    CONST robtarget rA_t486 := [[-156.188,32.3569,3418.1],[0.820893,-0.20476,-0.394721,0.358334],[1,0,2,0],[9E+09,9E+09,9E+09,9E+09,9E+09,9E+09]];
    CONST robtarget rB_t486 := [[608.123,552.232,3105.31],[0.872277,-0.183235,0.197016,-0.408341],[0,-2,0,0],[9E+09,9E+09,9E+09,9E+09,9E+09,9E+09]];
    CONST robtarget rB_t486_c5 := [[608.123,552.232,3105.31],[0.872277,-0.183235,0.197016,-0.408341],[0,0,0,0],[9E+09,9E+09,9E+09,9E+09,9E+09,9E+09]];
    CONST jointtarget jA_t486 := [[135,-13.9732,-69.2642,45,47.8597,225],[9E+09,9E+09,9E+09,9E+09,9E+09,9E+09]];
    CONST jointtarget jB_t486 := [[44.9992,-24.9745,-22.5996,-135.001,19.5471,44.9992],[9E+09,9E+09,9E+09,9E+09,9E+09,9E+09]];
    CONST jointtarget jBseed_t486 := [[44.9992,-24.9745,-22.5996,-135.001,19.5471,44.9992],[9E+09,9E+09,9E+09,9E+09,9E+09,9E+09]];

    CONST robtarget rA_t488 := [[-1759.7,-1640.61,1999.46],[0.855755,-0.00396172,-0.496397,0.145798],[-2,2,-1,0],[9E+09,9E+09,9E+09,9E+09,9E+09,9E+09]];
    CONST robtarget rB_t488 := [[478.399,-39.3809,2596.98],[0.780574,-0.0851872,0.494213,-0.373097],[-1,-1,-1,0],[9E+09,9E+09,9E+09,9E+09,9E+09,9E+09]];
    CONST robtarget rB_t488_c5 := [[478.399,-39.3809,2596.98],[0.780574,-0.0851872,0.494213,-0.373097],[0,0,0,0],[9E+09,9E+09,9E+09,9E+09,9E+09,9E+09]];
    CONST jointtarget jA_t488 := [[-135.001,22.0814,-22.3377,224.999,45.461,-45.001],[9E+09,9E+09,9E+09,9E+09,9E+09,9E+09]];
    CONST jointtarget jB_t488 := [[-0.000711459,-56.8981,12.0994,-45.0007,19.4775,-0.00071639],[9E+09,9E+09,9E+09,9E+09,9E+09,9E+09]];
    CONST jointtarget jBseed_t488 := [[-0.000711051,-56.8981,12.0994,-45.0007,19.4775,-0.000711051],[9E+09,9E+09,9E+09,9E+09,9E+09,9E+09]];

    CONST robtarget rA_t489 := [[478.399,-39.3809,2596.98],[0.780574,-0.0851872,0.494213,-0.373097],[-1,-1,-1,0],[9E+09,9E+09,9E+09,9E+09,9E+09,9E+09]];
    CONST robtarget rB_t489 := [[-73.1734,1033.07,3314.31],[0.0648344,0.215246,-0.280952,-0.933023],[1,-3,4,0],[9E+09,9E+09,9E+09,9E+09,9E+09,9E+09]];
    CONST robtarget rB_t489_c4 := [[-73.1734,1033.07,3314.31],[0.0648344,0.215246,-0.280952,-0.933023],[0,-4,0,0],[9E+09,9E+09,9E+09,9E+09,9E+09,9E+09]];
    CONST robtarget rB_t489_c5 := [[-73.1734,1033.07,3314.31],[0.0648344,0.215246,-0.280952,-0.933023],[0,0,0,0],[9E+09,9E+09,9E+09,9E+09,9E+09,9E+09]];
    CONST jointtarget jA_t489 := [[-0.000711459,-56.8981,12.0994,-45.0007,19.4775,-0.00071639],[9E+09,9E+09,9E+09,9E+09,9E+09,9E+09]];
    CONST jointtarget jB_t489 := [[90.0008,-2.94625,-53.5374,-269.999,25.9816,360.001],[9E+09,9E+09,9E+09,9E+09,9E+09,9E+09]];
    CONST jointtarget jBseed_t489 := [[90.0008,-2.94625,-53.5374,-269.999,25.9816,360.001],[9E+09,9E+09,9E+09,9E+09,9E+09,9E+09]];

    CONST robtarget rA_t490 := [[-73.1734,1033.07,3314.31],[0.0648344,0.215246,-0.280952,-0.933023],[1,-3,4,0],[9E+09,9E+09,9E+09,9E+09,9E+09,9E+09]];
    CONST robtarget rB_t490 := [[1761.71,1761.73,978.083],[0.626552,-0.67896,0.281238,-0.25952],[0,2,1,0],[9E+09,9E+09,9E+09,9E+09,9E+09,9E+09]];
    CONST robtarget rB_t490_c4 := [[1761.71,1761.73,978.083],[0.626552,-0.67896,0.281238,-0.25952],[0,-4,0,0],[9E+09,9E+09,9E+09,9E+09,9E+09,9E+09]];
    CONST jointtarget jA_t490 := [[90.0008,-2.94625,-53.5374,-269.999,25.9816,360.001],[9E+09,9E+09,9E+09,9E+09,9E+09,9E+09]];
    CONST jointtarget jB_t490 := [[45.0004,31.2076,0.22889,180,26.8386,90.0004],[9E+09,9E+09,9E+09,9E+09,9E+09,9E+09]];
    CONST jointtarget jBseed_t490 := [[45.0004,31.2076,0.228889,180,26.8386,90.0004],[9E+09,9E+09,9E+09,9E+09,9E+09,9E+09]];

    CONST robtarget rA_t491 := [[1761.71,1761.73,978.083],[0.626552,-0.67896,0.281238,-0.25952],[0,2,1,0],[9E+09,9E+09,9E+09,9E+09,9E+09,9E+09]];
    CONST robtarget rB_t491 := [[1223.98,-1223.96,143.412],[2.98331E-6,-0.66368,0.663686,-0.345034],[-1,-2,0,0],[9E+09,9E+09,9E+09,9E+09,9E+09,9E+09]];
    CONST robtarget rB_t491_c5 := [[1223.98,-1223.96,143.412],[2.98331E-6,-0.66368,0.663686,-0.345034],[0,0,0,0],[9E+09,9E+09,9E+09,9E+09,9E+09,9E+09]];
    CONST jointtarget jA_t491 := [[45.0004,31.2076,0.22889,180,26.8386,90.0004],[9E+09,9E+09,9E+09,9E+09,9E+09,9E+09]];
    CONST jointtarget jB_t491 := [[-44.9995,29.8453,38.9825,-180,19.1955,45.0005],[9E+09,9E+09,9E+09,9E+09,9E+09,9E+09]];
    CONST jointtarget jBseed_t491 := [[-44.9995,29.8453,38.9825,-180,19.1955,45.0005],[9E+09,9E+09,9E+09,9E+09,9E+09,9E+09]];

    CONST robtarget rA_t493 := [[-1447.52,-1512.75,2305.66],[0.839026,0.447646,-0.295573,0.091021],[-2,1,0,0],[9E+09,9E+09,9E+09,9E+09,9E+09,9E+09]];
    CONST robtarget rB_t493 := [[2344.51,-8.74922,2203.58],[0.526763,-0.443476,0.471721,-0.550753],[-1,3,4,0],[9E+09,9E+09,9E+09,9E+09,9E+09,9E+09]];
    CONST robtarget rB_t493_c3 := [[2344.51,-8.74922,2203.58],[0.526763,-0.443476,0.471721,-0.550753],[0,4,-4,0],[9E+09,9E+09,9E+09,9E+09,9E+09,9E+09]];
    CONST robtarget rB_t493_c8 := [[2344.51,-8.74922,2203.58],[0.526763,-0.443476,0.471721,-0.550753],[0,0,4,0],[9E+09,9E+09,9E+09,9E+09,9E+09,9E+09]];
    CONST jointtarget jA_t493 := [[-134.999,6.97836,-16.4937,135.001,22.9841,0.000509764],[9E+09,9E+09,9E+09,9E+09,9E+09,9E+09]];
    CONST jointtarget jB_t493 := [[-7.97153E-6,19.0307,-28.3444,270,3.00302,360],[9E+09,9E+09,9E+09,9E+09,9E+09,9E+09]];
    CONST jointtarget jBseed_t493 := [[-7.96537E-6,19.0307,-28.3444,270,3.00302,360],[9E+09,9E+09,9E+09,9E+09,9E+09,9E+09]];

    CONST robtarget rA_t495 := [[-0.00695535,-2301,2529.89],[0.361469,0.125634,0.30331,-0.872674],[-2,-3,-3,0],[9E+09,9E+09,9E+09,9E+09,9E+09,9E+09]];
    CONST robtarget rB_t495 := [[224.882,111.994,2748.59],[0.23447,0.140883,0.427482,0.861647],[0,-3,0,0],[9E+09,9E+09,9E+09,9E+09,9E+09,9E+09]];
    CONST robtarget rB_t495_c1 := [[224.882,111.994,2748.59],[0.23447,0.140883,0.427482,0.861647],[0,-4,-4,0],[9E+09,9E+09,9E+09,9E+09,9E+09,9E+09]];
    CONST robtarget rB_t495_c4 := [[224.882,111.994,2748.59],[0.23447,0.140883,0.427482,0.861647],[0,-4,0,0],[9E+09,9E+09,9E+09,9E+09,9E+09,9E+09]];
    CONST jointtarget jA_t495 := [[-90.0002,26.2526,-46.5508,-180,31.3706,-225],[9E+09,9E+09,9E+09,9E+09,9E+09,9E+09]];
    CONST jointtarget jB_t495 := [[0.000893293,-56.455,3.14889,-269.999,42.1137,45.0009],[9E+09,9E+09,9E+09,9E+09,9E+09,9E+09]];
    CONST jointtarget jBseed_t495 := [[0.000892148,-56.455,3.1489,-269.999,42.1137,45.0009],[9E+09,9E+09,9E+09,9E+09,9E+09,9E+09]];

    CONST robtarget rA_t496 := [[224.882,111.994,2748.59],[0.23447,0.140883,0.427482,0.861647],[0,-3,0,0],[9E+09,9E+09,9E+09,9E+09,9E+09,9E+09]];
    CONST robtarget rB_t496 := [[1431.74,-1585.91,602.66],[0.322926,0.522416,-0.706832,0.350983],[-1,3,-1,0],[9E+09,9E+09,9E+09,9E+09,9E+09,9E+09]];
    CONST robtarget rB_t496_c5 := [[1431.74,-1585.91,602.66],[0.322926,0.522416,-0.706832,0.350983],[0,0,0,0],[9E+09,9E+09,9E+09,9E+09,9E+09,9E+09]];
    CONST jointtarget jA_t496 := [[0.000893293,-56.455,3.14889,-269.999,42.1137,45.0009],[9E+09,9E+09,9E+09,9E+09,9E+09,9E+09]];
    CONST jointtarget jB_t496 := [[-44.9994,26.9448,19.078,270.001,40.7624,-44.9994],[9E+09,9E+09,9E+09,9E+09,9E+09,9E+09]];
    CONST jointtarget jBseed_t496 := [[-44.9994,26.9448,19.078,270.001,40.7624,-44.9994],[9E+09,9E+09,9E+09,9E+09,9E+09,9E+09]];

    CONST robtarget rA_t498 := [[-1697.1,1644.42,846.92],[0.0841501,-0.833571,0.288989,0.46321],[1,0,-2,0],[9E+09,9E+09,9E+09,9E+09,9E+09,9E+09]];
    CONST robtarget rB_t498 := [[2209.47,38.6604,2536.25],[0.374617,-0.554189,0.125353,-0.732682],[-1,0,1,0],[9E+09,9E+09,9E+09,9E+09,9E+09,9E+09]];
    CONST robtarget rB_t498_c2 := [[2209.47,38.6604,2536.25],[0.374617,-0.554189,0.125353,-0.732682],[0,0,-4,0],[9E+09,9E+09,9E+09,9E+09,9E+09,9E+09]];
    CONST jointtarget jA_t498 := [[134.999,27.9336,6.89413,89.9995,12.8947,-90.0005],[9E+09,9E+09,9E+09,9E+09,9E+09,9E+09]];
    CONST jointtarget jB_t498 := [[-0.000138064,19.2798,-40.6394,89.9999,13.3872,135],[9E+09,9E+09,9E+09,9E+09,9E+09,9E+09]];
    CONST jointtarget jBseed_t498 := [[-0.000138096,19.2798,-40.6394,89.9999,13.3872,135],[9E+09,9E+09,9E+09,9E+09,9E+09,9E+09]];

    ! B* configuration values by successful test/conf
    CONST num bStarCf1_t1_c5 := 0;
    CONST num bStarCf4_t1_c5 := 0;
    CONST num bStarCf6_t1_c5 := 0;
    CONST num bStarCfx_t1_c5 := 0;

    CONST num bStarCf1_t1_c6 := 0;
    CONST num bStarCf4_t1_c6 := 4;
    CONST num bStarCf6_t1_c6 := 0;
    CONST num bStarCfx_t1_c6 := 0;

    CONST num bStarCf1_t4_c1 := 0;
    CONST num bStarCf4_t4_c1 := -4;
    CONST num bStarCf6_t4_c1 := -4;
    CONST num bStarCfx_t4_c1 := 0;

    CONST num bStarCf1_t4_c4 := 0;
    CONST num bStarCf4_t4_c4 := -4;
    CONST num bStarCf6_t4_c4 := 0;
    CONST num bStarCfx_t4_c4 := 0;

    CONST num bStarCf1_t7_c1 := 0;
    CONST num bStarCf4_t7_c1 := -4;
    CONST num bStarCf6_t7_c1 := -4;
    CONST num bStarCfx_t7_c1 := 0;

    CONST num bStarCf1_t7_c2 := 0;
    CONST num bStarCf4_t7_c2 := 0;
    CONST num bStarCf6_t7_c2 := -4;
    CONST num bStarCfx_t7_c2 := 0;

    CONST num bStarCf1_t9_c5 := 0;
    CONST num bStarCf4_t9_c5 := 0;
    CONST num bStarCf6_t9_c5 := 0;
    CONST num bStarCfx_t9_c5 := 0;

    CONST num bStarCf1_t12_c4 := 0;
    CONST num bStarCf4_t12_c4 := -4;
    CONST num bStarCf6_t12_c4 := 0;
    CONST num bStarCfx_t12_c4 := 0;

    CONST num bStarCf1_t12_c5 := 0;
    CONST num bStarCf4_t12_c5 := 0;
    CONST num bStarCf6_t12_c5 := 0;
    CONST num bStarCfx_t12_c5 := 0;

    CONST num bStarCf1_t16_c2 := 0;
    CONST num bStarCf4_t16_c2 := 0;
    CONST num bStarCf6_t16_c2 := -4;
    CONST num bStarCfx_t16_c2 := 0;

    CONST num bStarCf1_t19_c2 := 0;
    CONST num bStarCf4_t19_c2 := 0;
    CONST num bStarCf6_t19_c2 := -4;
    CONST num bStarCfx_t19_c2 := 0;

    CONST num bStarCf1_t22_c5 := 0;
    CONST num bStarCf4_t22_c5 := 0;
    CONST num bStarCf6_t22_c5 := 0;
    CONST num bStarCfx_t22_c5 := 0;

    CONST num bStarCf1_t23_c6 := 0;
    CONST num bStarCf4_t23_c6 := 4;
    CONST num bStarCf6_t23_c6 := 0;
    CONST num bStarCfx_t23_c6 := 0;

    CONST num bStarCf1_t27_c5 := 0;
    CONST num bStarCf4_t27_c5 := 0;
    CONST num bStarCf6_t27_c5 := 0;
    CONST num bStarCfx_t27_c5 := 0;

    CONST num bStarCf1_t27_c8 := 0;
    CONST num bStarCf4_t27_c8 := 0;
    CONST num bStarCf6_t27_c8 := 4;
    CONST num bStarCfx_t27_c8 := 0;

    CONST num bStarCf1_t28_c5 := 0;
    CONST num bStarCf4_t28_c5 := 0;
    CONST num bStarCf6_t28_c5 := 0;
    CONST num bStarCfx_t28_c5 := 0;

    CONST num bStarCf1_t31_c1 := 0;
    CONST num bStarCf4_t31_c1 := -4;
    CONST num bStarCf6_t31_c1 := -4;
    CONST num bStarCfx_t31_c1 := 0;

    CONST num bStarCf1_t31_c4 := 0;
    CONST num bStarCf4_t31_c4 := -4;
    CONST num bStarCf6_t31_c4 := 0;
    CONST num bStarCfx_t31_c4 := 0;

    CONST num bStarCf1_t37_c5 := 0;
    CONST num bStarCf4_t37_c5 := 0;
    CONST num bStarCf6_t37_c5 := 0;
    CONST num bStarCfx_t37_c5 := 0;

    CONST num bStarCf1_t40_c8 := 0;
    CONST num bStarCf4_t40_c8 := 0;
    CONST num bStarCf6_t40_c8 := 4;
    CONST num bStarCfx_t40_c8 := 0;

    CONST num bStarCf1_t46_c1 := 0;
    CONST num bStarCf4_t46_c1 := -4;
    CONST num bStarCf6_t46_c1 := -4;
    CONST num bStarCfx_t46_c1 := 0;

    CONST num bStarCf1_t46_c2 := 0;
    CONST num bStarCf4_t46_c2 := 0;
    CONST num bStarCf6_t46_c2 := -4;
    CONST num bStarCfx_t46_c2 := 0;

    CONST num bStarCf1_t50_c7 := 0;
    CONST num bStarCf4_t50_c7 := -4;
    CONST num bStarCf6_t50_c7 := 4;
    CONST num bStarCfx_t50_c7 := 0;

    CONST num bStarCf1_t51_c5 := 0;
    CONST num bStarCf4_t51_c5 := 0;
    CONST num bStarCf6_t51_c5 := 0;
    CONST num bStarCfx_t51_c5 := 0;

    CONST num bStarCf1_t51_c8 := 0;
    CONST num bStarCf4_t51_c8 := 0;
    CONST num bStarCf6_t51_c8 := 4;
    CONST num bStarCfx_t51_c8 := 0;

    CONST num bStarCf1_t53_c1 := 0;
    CONST num bStarCf4_t53_c1 := -4;
    CONST num bStarCf6_t53_c1 := -4;
    CONST num bStarCfx_t53_c1 := 0;

    CONST num bStarCf1_t56_c2 := 0;
    CONST num bStarCf4_t56_c2 := 0;
    CONST num bStarCf6_t56_c2 := -4;
    CONST num bStarCfx_t56_c2 := 0;

    CONST num bStarCf1_t56_c5 := 0;
    CONST num bStarCf4_t56_c5 := 0;
    CONST num bStarCf6_t56_c5 := 0;
    CONST num bStarCfx_t56_c5 := 0;

    CONST num bStarCf1_t58_c8 := 0;
    CONST num bStarCf4_t58_c8 := 0;
    CONST num bStarCf6_t58_c8 := 4;
    CONST num bStarCfx_t58_c8 := 0;

    CONST num bStarCf1_t64_c4 := 0;
    CONST num bStarCf4_t64_c4 := -4;
    CONST num bStarCf6_t64_c4 := 0;
    CONST num bStarCfx_t64_c4 := 0;

    CONST num bStarCf1_t66_c4 := 0;
    CONST num bStarCf4_t66_c4 := -4;
    CONST num bStarCf6_t66_c4 := 0;
    CONST num bStarCfx_t66_c4 := 0;

    CONST num bStarCf1_t67_c2 := 0;
    CONST num bStarCf4_t67_c2 := 0;
    CONST num bStarCf6_t67_c2 := -4;
    CONST num bStarCfx_t67_c2 := 0;

    CONST num bStarCf1_t67_c3 := 0;
    CONST num bStarCf4_t67_c3 := 4;
    CONST num bStarCf6_t67_c3 := -4;
    CONST num bStarCfx_t67_c3 := 0;

    CONST num bStarCf1_t68_c4 := 0;
    CONST num bStarCf4_t68_c4 := -4;
    CONST num bStarCf6_t68_c4 := 0;
    CONST num bStarCfx_t68_c4 := 0;

    CONST num bStarCf1_t69_c4 := 0;
    CONST num bStarCf4_t69_c4 := -4;
    CONST num bStarCf6_t69_c4 := 0;
    CONST num bStarCfx_t69_c4 := 0;

    CONST num bStarCf1_t72_c5 := 0;
    CONST num bStarCf4_t72_c5 := 0;
    CONST num bStarCf6_t72_c5 := 0;
    CONST num bStarCfx_t72_c5 := 0;

    CONST num bStarCf1_t73_c4 := 0;
    CONST num bStarCf4_t73_c4 := -4;
    CONST num bStarCf6_t73_c4 := 0;
    CONST num bStarCfx_t73_c4 := 0;

    CONST num bStarCf1_t74_c4 := 0;
    CONST num bStarCf4_t74_c4 := -4;
    CONST num bStarCf6_t74_c4 := 0;
    CONST num bStarCfx_t74_c4 := 0;

    CONST num bStarCf1_t79_c1 := 0;
    CONST num bStarCf4_t79_c1 := -4;
    CONST num bStarCf6_t79_c1 := -4;
    CONST num bStarCfx_t79_c1 := 0;

    CONST num bStarCf1_t79_c4 := 0;
    CONST num bStarCf4_t79_c4 := -4;
    CONST num bStarCf6_t79_c4 := 0;
    CONST num bStarCfx_t79_c4 := 0;

    CONST num bStarCf1_t82_c8 := 0;
    CONST num bStarCf4_t82_c8 := 0;
    CONST num bStarCf6_t82_c8 := 4;
    CONST num bStarCfx_t82_c8 := 0;

    CONST num bStarCf1_t82_c9 := 0;
    CONST num bStarCf4_t82_c9 := 4;
    CONST num bStarCf6_t82_c9 := 4;
    CONST num bStarCfx_t82_c9 := 0;

    CONST num bStarCf1_t83_c5 := 0;
    CONST num bStarCf4_t83_c5 := 0;
    CONST num bStarCf6_t83_c5 := 0;
    CONST num bStarCfx_t83_c5 := 0;

    CONST num bStarCf1_t83_c8 := 0;
    CONST num bStarCf4_t83_c8 := 0;
    CONST num bStarCf6_t83_c8 := 4;
    CONST num bStarCfx_t83_c8 := 0;

    CONST num bStarCf1_t85_c8 := 0;
    CONST num bStarCf4_t85_c8 := 0;
    CONST num bStarCf6_t85_c8 := 4;
    CONST num bStarCfx_t85_c8 := 0;

    CONST num bStarCf1_t88_c5 := 0;
    CONST num bStarCf4_t88_c5 := 0;
    CONST num bStarCf6_t88_c5 := 0;
    CONST num bStarCfx_t88_c5 := 0;

    CONST num bStarCf1_t89_c5 := 0;
    CONST num bStarCf4_t89_c5 := 0;
    CONST num bStarCf6_t89_c5 := 0;
    CONST num bStarCfx_t89_c5 := 0;

    CONST num bStarCf1_t90_c5 := 0;
    CONST num bStarCf4_t90_c5 := 0;
    CONST num bStarCf6_t90_c5 := 0;
    CONST num bStarCfx_t90_c5 := 0;

    CONST num bStarCf1_t102_c3 := 0;
    CONST num bStarCf4_t102_c3 := 4;
    CONST num bStarCf6_t102_c3 := -4;
    CONST num bStarCfx_t102_c3 := 0;

    CONST num bStarCf1_t103_c5 := 0;
    CONST num bStarCf4_t103_c5 := 0;
    CONST num bStarCf6_t103_c5 := 0;
    CONST num bStarCfx_t103_c5 := 0;

    CONST num bStarCf1_t104_c1 := 0;
    CONST num bStarCf4_t104_c1 := -4;
    CONST num bStarCf6_t104_c1 := -4;
    CONST num bStarCfx_t104_c1 := 0;

    CONST num bStarCf1_t107_c5 := 0;
    CONST num bStarCf4_t107_c5 := 0;
    CONST num bStarCf6_t107_c5 := 0;
    CONST num bStarCfx_t107_c5 := 0;

    CONST num bStarCf1_t108_c2 := 0;
    CONST num bStarCf4_t108_c2 := 0;
    CONST num bStarCf6_t108_c2 := -4;
    CONST num bStarCfx_t108_c2 := 0;

    CONST num bStarCf1_t108_c3 := 0;
    CONST num bStarCf4_t108_c3 := 4;
    CONST num bStarCf6_t108_c3 := -4;
    CONST num bStarCfx_t108_c3 := 0;

    CONST num bStarCf1_t109_c6 := 0;
    CONST num bStarCf4_t109_c6 := 4;
    CONST num bStarCf6_t109_c6 := 0;
    CONST num bStarCfx_t109_c6 := 0;

    CONST num bStarCf1_t110_c2 := 0;
    CONST num bStarCf4_t110_c2 := 0;
    CONST num bStarCf6_t110_c2 := -4;
    CONST num bStarCfx_t110_c2 := 0;

    CONST num bStarCf1_t111_c5 := 0;
    CONST num bStarCf4_t111_c5 := 0;
    CONST num bStarCf6_t111_c5 := 0;
    CONST num bStarCfx_t111_c5 := 0;

    CONST num bStarCf1_t111_c8 := 0;
    CONST num bStarCf4_t111_c8 := 0;
    CONST num bStarCf6_t111_c8 := 4;
    CONST num bStarCfx_t111_c8 := 0;

    CONST num bStarCf1_t115_c4 := 0;
    CONST num bStarCf4_t115_c4 := -4;
    CONST num bStarCf6_t115_c4 := 0;
    CONST num bStarCfx_t115_c4 := 0;

    CONST num bStarCf1_t115_c5 := 0;
    CONST num bStarCf4_t115_c5 := 0;
    CONST num bStarCf6_t115_c5 := 0;
    CONST num bStarCfx_t115_c5 := 0;

    CONST num bStarCf1_t116_c2 := 0;
    CONST num bStarCf4_t116_c2 := 0;
    CONST num bStarCf6_t116_c2 := -4;
    CONST num bStarCfx_t116_c2 := 0;

    CONST num bStarCf1_t116_c5 := 0;
    CONST num bStarCf4_t116_c5 := 0;
    CONST num bStarCf6_t116_c5 := 0;
    CONST num bStarCfx_t116_c5 := 0;

    CONST num bStarCf1_t117_c7 := 0;
    CONST num bStarCf4_t117_c7 := -4;
    CONST num bStarCf6_t117_c7 := 4;
    CONST num bStarCfx_t117_c7 := 0;

    CONST num bStarCf1_t119_c1 := 0;
    CONST num bStarCf4_t119_c1 := -4;
    CONST num bStarCf6_t119_c1 := -4;
    CONST num bStarCfx_t119_c1 := 0;

    CONST num bStarCf1_t122_c1 := 0;
    CONST num bStarCf4_t122_c1 := -4;
    CONST num bStarCf6_t122_c1 := -4;
    CONST num bStarCfx_t122_c1 := 0;

    CONST num bStarCf1_t122_c2 := 0;
    CONST num bStarCf4_t122_c2 := 0;
    CONST num bStarCf6_t122_c2 := -4;
    CONST num bStarCfx_t122_c2 := 0;

    CONST num bStarCf1_t124_c5 := 0;
    CONST num bStarCf4_t124_c5 := 0;
    CONST num bStarCf6_t124_c5 := 0;
    CONST num bStarCfx_t124_c5 := 0;

    CONST num bStarCf1_t126_c5 := 0;
    CONST num bStarCf4_t126_c5 := 0;
    CONST num bStarCf6_t126_c5 := 0;
    CONST num bStarCfx_t126_c5 := 0;

    CONST num bStarCf1_t129_c4 := 0;
    CONST num bStarCf4_t129_c4 := -4;
    CONST num bStarCf6_t129_c4 := 0;
    CONST num bStarCfx_t129_c4 := 0;

    CONST num bStarCf1_t129_c5 := 0;
    CONST num bStarCf4_t129_c5 := 0;
    CONST num bStarCf6_t129_c5 := 0;
    CONST num bStarCfx_t129_c5 := 0;

    CONST num bStarCf1_t131_c4 := 0;
    CONST num bStarCf4_t131_c4 := -4;
    CONST num bStarCf6_t131_c4 := 0;
    CONST num bStarCfx_t131_c4 := 0;

    CONST num bStarCf1_t133_c2 := 0;
    CONST num bStarCf4_t133_c2 := 0;
    CONST num bStarCf6_t133_c2 := -4;
    CONST num bStarCfx_t133_c2 := 0;

    CONST num bStarCf1_t134_c2 := 0;
    CONST num bStarCf4_t134_c2 := 0;
    CONST num bStarCf6_t134_c2 := -4;
    CONST num bStarCfx_t134_c2 := 0;

    CONST num bStarCf1_t134_c5 := 0;
    CONST num bStarCf4_t134_c5 := 0;
    CONST num bStarCf6_t134_c5 := 0;
    CONST num bStarCfx_t134_c5 := 0;

    CONST num bStarCf1_t142_c5 := 0;
    CONST num bStarCf4_t142_c5 := 0;
    CONST num bStarCf6_t142_c5 := 0;
    CONST num bStarCfx_t142_c5 := 0;

    CONST num bStarCf1_t143_c5 := 0;
    CONST num bStarCf4_t143_c5 := 0;
    CONST num bStarCf6_t143_c5 := 0;
    CONST num bStarCfx_t143_c5 := 0;

    CONST num bStarCf1_t149_c5 := 0;
    CONST num bStarCf4_t149_c5 := 0;
    CONST num bStarCf6_t149_c5 := 0;
    CONST num bStarCfx_t149_c5 := 0;

    CONST num bStarCf1_t152_c8 := 0;
    CONST num bStarCf4_t152_c8 := 0;
    CONST num bStarCf6_t152_c8 := 4;
    CONST num bStarCfx_t152_c8 := 0;

    CONST num bStarCf1_t153_c5 := 0;
    CONST num bStarCf4_t153_c5 := 0;
    CONST num bStarCf6_t153_c5 := 0;
    CONST num bStarCfx_t153_c5 := 0;

    CONST num bStarCf1_t154_c5 := 0;
    CONST num bStarCf4_t154_c5 := 0;
    CONST num bStarCf6_t154_c5 := 0;
    CONST num bStarCfx_t154_c5 := 0;

    CONST num bStarCf1_t157_c8 := 0;
    CONST num bStarCf4_t157_c8 := 0;
    CONST num bStarCf6_t157_c8 := 4;
    CONST num bStarCfx_t157_c8 := 0;

    CONST num bStarCf1_t159_c4 := 0;
    CONST num bStarCf4_t159_c4 := -4;
    CONST num bStarCf6_t159_c4 := 0;
    CONST num bStarCfx_t159_c4 := 0;

    CONST num bStarCf1_t163_c5 := 0;
    CONST num bStarCf4_t163_c5 := 0;
    CONST num bStarCf6_t163_c5 := 0;
    CONST num bStarCfx_t163_c5 := 0;

    CONST num bStarCf1_t165_c3 := 0;
    CONST num bStarCf4_t165_c3 := 4;
    CONST num bStarCf6_t165_c3 := -4;
    CONST num bStarCfx_t165_c3 := 0;

    CONST num bStarCf1_t165_c6 := 0;
    CONST num bStarCf4_t165_c6 := 4;
    CONST num bStarCf6_t165_c6 := 0;
    CONST num bStarCfx_t165_c6 := 0;

    CONST num bStarCf1_t166_c5 := 0;
    CONST num bStarCf4_t166_c5 := 0;
    CONST num bStarCf6_t166_c5 := 0;
    CONST num bStarCfx_t166_c5 := 0;

    CONST num bStarCf1_t167_c2 := 0;
    CONST num bStarCf4_t167_c2 := 0;
    CONST num bStarCf6_t167_c2 := -4;
    CONST num bStarCfx_t167_c2 := 0;

    CONST num bStarCf1_t167_c5 := 0;
    CONST num bStarCf4_t167_c5 := 0;
    CONST num bStarCf6_t167_c5 := 0;
    CONST num bStarCfx_t167_c5 := 0;

    CONST num bStarCf1_t170_c4 := 0;
    CONST num bStarCf4_t170_c4 := -4;
    CONST num bStarCf6_t170_c4 := 0;
    CONST num bStarCfx_t170_c4 := 0;

    CONST num bStarCf1_t171_c4 := 0;
    CONST num bStarCf4_t171_c4 := -4;
    CONST num bStarCf6_t171_c4 := 0;
    CONST num bStarCfx_t171_c4 := 0;

    CONST num bStarCf1_t171_c5 := 0;
    CONST num bStarCf4_t171_c5 := 0;
    CONST num bStarCf6_t171_c5 := 0;
    CONST num bStarCfx_t171_c5 := 0;

    CONST num bStarCf1_t174_c3 := 0;
    CONST num bStarCf4_t174_c3 := 4;
    CONST num bStarCf6_t174_c3 := -4;
    CONST num bStarCfx_t174_c3 := 0;

    CONST num bStarCf1_t177_c1 := 0;
    CONST num bStarCf4_t177_c1 := -4;
    CONST num bStarCf6_t177_c1 := -4;
    CONST num bStarCfx_t177_c1 := 0;

    CONST num bStarCf1_t183_c2 := 0;
    CONST num bStarCf4_t183_c2 := 0;
    CONST num bStarCf6_t183_c2 := -4;
    CONST num bStarCfx_t183_c2 := 0;

    CONST num bStarCf1_t183_c5 := 0;
    CONST num bStarCf4_t183_c5 := 0;
    CONST num bStarCf6_t183_c5 := 0;
    CONST num bStarCfx_t183_c5 := 0;

    CONST num bStarCf1_t187_c6 := 0;
    CONST num bStarCf4_t187_c6 := 4;
    CONST num bStarCf6_t187_c6 := 0;
    CONST num bStarCfx_t187_c6 := 0;

    CONST num bStarCf1_t188_c2 := 0;
    CONST num bStarCf4_t188_c2 := 0;
    CONST num bStarCf6_t188_c2 := -4;
    CONST num bStarCfx_t188_c2 := 0;

    CONST num bStarCf1_t192_c2 := 0;
    CONST num bStarCf4_t192_c2 := 0;
    CONST num bStarCf6_t192_c2 := -4;
    CONST num bStarCfx_t192_c2 := 0;

    CONST num bStarCf1_t194_c5 := 0;
    CONST num bStarCf4_t194_c5 := 0;
    CONST num bStarCf6_t194_c5 := 0;
    CONST num bStarCfx_t194_c5 := 0;

    CONST num bStarCf1_t195_c5 := 0;
    CONST num bStarCf4_t195_c5 := 0;
    CONST num bStarCf6_t195_c5 := 0;
    CONST num bStarCfx_t195_c5 := 0;

    CONST num bStarCf1_t197_c4 := 0;
    CONST num bStarCf4_t197_c4 := -4;
    CONST num bStarCf6_t197_c4 := 0;
    CONST num bStarCfx_t197_c4 := 0;

    CONST num bStarCf1_t198_c2 := 0;
    CONST num bStarCf4_t198_c2 := 0;
    CONST num bStarCf6_t198_c2 := -4;
    CONST num bStarCfx_t198_c2 := 0;

    CONST num bStarCf1_t198_c3 := 0;
    CONST num bStarCf4_t198_c3 := 4;
    CONST num bStarCf6_t198_c3 := -4;
    CONST num bStarCfx_t198_c3 := 0;

    CONST num bStarCf1_t200_c2 := 0;
    CONST num bStarCf4_t200_c2 := 0;
    CONST num bStarCf6_t200_c2 := -4;
    CONST num bStarCfx_t200_c2 := 0;

    CONST num bStarCf1_t205_c6 := 0;
    CONST num bStarCf4_t205_c6 := 4;
    CONST num bStarCf6_t205_c6 := 0;
    CONST num bStarCfx_t205_c6 := 0;

    CONST num bStarCf1_t207_c5 := 0;
    CONST num bStarCf4_t207_c5 := 0;
    CONST num bStarCf6_t207_c5 := 0;
    CONST num bStarCfx_t207_c5 := 0;

    CONST num bStarCf1_t208_c2 := 0;
    CONST num bStarCf4_t208_c2 := 0;
    CONST num bStarCf6_t208_c2 := -4;
    CONST num bStarCfx_t208_c2 := 0;

    CONST num bStarCf1_t210_c4 := 0;
    CONST num bStarCf4_t210_c4 := -4;
    CONST num bStarCf6_t210_c4 := 0;
    CONST num bStarCfx_t210_c4 := 0;

    CONST num bStarCf1_t210_c7 := 0;
    CONST num bStarCf4_t210_c7 := -4;
    CONST num bStarCf6_t210_c7 := 4;
    CONST num bStarCfx_t210_c7 := 0;

    CONST num bStarCf1_t213_c2 := 0;
    CONST num bStarCf4_t213_c2 := 0;
    CONST num bStarCf6_t213_c2 := -4;
    CONST num bStarCfx_t213_c2 := 0;

    CONST num bStarCf1_t215_c4 := 0;
    CONST num bStarCf4_t215_c4 := -4;
    CONST num bStarCf6_t215_c4 := 0;
    CONST num bStarCfx_t215_c4 := 0;

    CONST num bStarCf1_t216_c4 := 0;
    CONST num bStarCf4_t216_c4 := -4;
    CONST num bStarCf6_t216_c4 := 0;
    CONST num bStarCfx_t216_c4 := 0;

    CONST num bStarCf1_t217_c5 := 0;
    CONST num bStarCf4_t217_c5 := 0;
    CONST num bStarCf6_t217_c5 := 0;
    CONST num bStarCfx_t217_c5 := 0;

    CONST num bStarCf1_t218_c5 := 0;
    CONST num bStarCf4_t218_c5 := 0;
    CONST num bStarCf6_t218_c5 := 0;
    CONST num bStarCfx_t218_c5 := 0;

    CONST num bStarCf1_t220_c5 := 0;
    CONST num bStarCf4_t220_c5 := 0;
    CONST num bStarCf6_t220_c5 := 0;
    CONST num bStarCfx_t220_c5 := 0;

    CONST num bStarCf1_t221_c6 := 0;
    CONST num bStarCf4_t221_c6 := 4;
    CONST num bStarCf6_t221_c6 := 0;
    CONST num bStarCfx_t221_c6 := 0;

    CONST num bStarCf1_t224_c8 := 0;
    CONST num bStarCf4_t224_c8 := 0;
    CONST num bStarCf6_t224_c8 := 4;
    CONST num bStarCfx_t224_c8 := 0;

    CONST num bStarCf1_t225_c5 := 0;
    CONST num bStarCf4_t225_c5 := 0;
    CONST num bStarCf6_t225_c5 := 0;
    CONST num bStarCfx_t225_c5 := 0;

    CONST num bStarCf1_t227_c2 := 0;
    CONST num bStarCf4_t227_c2 := 0;
    CONST num bStarCf6_t227_c2 := -4;
    CONST num bStarCfx_t227_c2 := 0;

    CONST num bStarCf1_t228_c5 := 0;
    CONST num bStarCf4_t228_c5 := 0;
    CONST num bStarCf6_t228_c5 := 0;
    CONST num bStarCfx_t228_c5 := 0;

    CONST num bStarCf1_t229_c9 := 0;
    CONST num bStarCf4_t229_c9 := 4;
    CONST num bStarCf6_t229_c9 := 4;
    CONST num bStarCfx_t229_c9 := 0;

    CONST num bStarCf1_t230_c5 := 0;
    CONST num bStarCf4_t230_c5 := 0;
    CONST num bStarCf6_t230_c5 := 0;
    CONST num bStarCfx_t230_c5 := 0;

    CONST num bStarCf1_t231_c5 := 0;
    CONST num bStarCf4_t231_c5 := 0;
    CONST num bStarCf6_t231_c5 := 0;
    CONST num bStarCfx_t231_c5 := 0;

    CONST num bStarCf1_t234_c2 := 0;
    CONST num bStarCf4_t234_c2 := 0;
    CONST num bStarCf6_t234_c2 := -4;
    CONST num bStarCfx_t234_c2 := 0;

    CONST num bStarCf1_t235_c2 := 0;
    CONST num bStarCf4_t235_c2 := 0;
    CONST num bStarCf6_t235_c2 := -4;
    CONST num bStarCfx_t235_c2 := 0;

    CONST num bStarCf1_t235_c5 := 0;
    CONST num bStarCf4_t235_c5 := 0;
    CONST num bStarCf6_t235_c5 := 0;
    CONST num bStarCfx_t235_c5 := 0;

    CONST num bStarCf1_t236_c2 := 0;
    CONST num bStarCf4_t236_c2 := 0;
    CONST num bStarCf6_t236_c2 := -4;
    CONST num bStarCfx_t236_c2 := 0;

    CONST num bStarCf1_t237_c5 := 0;
    CONST num bStarCf4_t237_c5 := 0;
    CONST num bStarCf6_t237_c5 := 0;
    CONST num bStarCfx_t237_c5 := 0;

    CONST num bStarCf1_t238_c5 := 0;
    CONST num bStarCf4_t238_c5 := 0;
    CONST num bStarCf6_t238_c5 := 0;
    CONST num bStarCfx_t238_c5 := 0;

    CONST num bStarCf1_t246_c7 := 0;
    CONST num bStarCf4_t246_c7 := -4;
    CONST num bStarCf6_t246_c7 := 4;
    CONST num bStarCfx_t246_c7 := 0;

    CONST num bStarCf1_t247_c5 := 0;
    CONST num bStarCf4_t247_c5 := 0;
    CONST num bStarCf6_t247_c5 := 0;
    CONST num bStarCfx_t247_c5 := 0;

    CONST num bStarCf1_t248_c4 := 0;
    CONST num bStarCf4_t248_c4 := -4;
    CONST num bStarCf6_t248_c4 := 0;
    CONST num bStarCfx_t248_c4 := 0;

    CONST num bStarCf1_t250_c5 := 0;
    CONST num bStarCf4_t250_c5 := 0;
    CONST num bStarCf6_t250_c5 := 0;
    CONST num bStarCfx_t250_c5 := 0;

    CONST num bStarCf1_t250_c8 := 0;
    CONST num bStarCf4_t250_c8 := 0;
    CONST num bStarCf6_t250_c8 := 4;
    CONST num bStarCfx_t250_c8 := 0;

    CONST num bStarCf1_t251_c4 := 0;
    CONST num bStarCf4_t251_c4 := -4;
    CONST num bStarCf6_t251_c4 := 0;
    CONST num bStarCfx_t251_c4 := 0;

    CONST num bStarCf1_t252_c7 := 0;
    CONST num bStarCf4_t252_c7 := -4;
    CONST num bStarCf6_t252_c7 := 4;
    CONST num bStarCfx_t252_c7 := 0;

    CONST num bStarCf1_t254_c5 := 0;
    CONST num bStarCf4_t254_c5 := 0;
    CONST num bStarCf6_t254_c5 := 0;
    CONST num bStarCfx_t254_c5 := 0;

    CONST num bStarCf1_t254_c8 := 0;
    CONST num bStarCf4_t254_c8 := 0;
    CONST num bStarCf6_t254_c8 := 4;
    CONST num bStarCfx_t254_c8 := 0;

    CONST num bStarCf1_t261_c5 := 0;
    CONST num bStarCf4_t261_c5 := 0;
    CONST num bStarCf6_t261_c5 := 0;
    CONST num bStarCfx_t261_c5 := 0;

    CONST num bStarCf1_t263_c2 := 0;
    CONST num bStarCf4_t263_c2 := 0;
    CONST num bStarCf6_t263_c2 := -4;
    CONST num bStarCfx_t263_c2 := 0;

    CONST num bStarCf1_t263_c5 := 0;
    CONST num bStarCf4_t263_c5 := 0;
    CONST num bStarCf6_t263_c5 := 0;
    CONST num bStarCfx_t263_c5 := 0;

    CONST num bStarCf1_t264_c4 := 0;
    CONST num bStarCf4_t264_c4 := -4;
    CONST num bStarCf6_t264_c4 := 0;
    CONST num bStarCfx_t264_c4 := 0;

    CONST num bStarCf1_t265_c5 := 0;
    CONST num bStarCf4_t265_c5 := 0;
    CONST num bStarCf6_t265_c5 := 0;
    CONST num bStarCfx_t265_c5 := 0;

    CONST num bStarCf1_t267_c7 := 0;
    CONST num bStarCf4_t267_c7 := -4;
    CONST num bStarCf6_t267_c7 := 4;
    CONST num bStarCfx_t267_c7 := 0;

    CONST num bStarCf1_t268_c5 := 0;
    CONST num bStarCf4_t268_c5 := 0;
    CONST num bStarCf6_t268_c5 := 0;
    CONST num bStarCfx_t268_c5 := 0;

    CONST num bStarCf1_t278_c1 := 0;
    CONST num bStarCf4_t278_c1 := -4;
    CONST num bStarCf6_t278_c1 := -4;
    CONST num bStarCfx_t278_c1 := 0;

    CONST num bStarCf1_t278_c2 := 0;
    CONST num bStarCf4_t278_c2 := 0;
    CONST num bStarCf6_t278_c2 := -4;
    CONST num bStarCfx_t278_c2 := 0;

    CONST num bStarCf1_t279_c4 := 0;
    CONST num bStarCf4_t279_c4 := -4;
    CONST num bStarCf6_t279_c4 := 0;
    CONST num bStarCfx_t279_c4 := 0;

    CONST num bStarCf1_t279_c7 := 0;
    CONST num bStarCf4_t279_c7 := -4;
    CONST num bStarCf6_t279_c7 := 4;
    CONST num bStarCfx_t279_c7 := 0;

    CONST num bStarCf1_t280_c1 := 0;
    CONST num bStarCf4_t280_c1 := -4;
    CONST num bStarCf6_t280_c1 := -4;
    CONST num bStarCfx_t280_c1 := 0;

    CONST num bStarCf1_t280_c2 := 0;
    CONST num bStarCf4_t280_c2 := 0;
    CONST num bStarCf6_t280_c2 := -4;
    CONST num bStarCfx_t280_c2 := 0;

    CONST num bStarCf1_t281_c5 := 0;
    CONST num bStarCf4_t281_c5 := 0;
    CONST num bStarCf6_t281_c5 := 0;
    CONST num bStarCfx_t281_c5 := 0;

    CONST num bStarCf1_t283_c5 := 0;
    CONST num bStarCf4_t283_c5 := 0;
    CONST num bStarCf6_t283_c5 := 0;
    CONST num bStarCfx_t283_c5 := 0;

    CONST num bStarCf1_t283_c8 := 0;
    CONST num bStarCf4_t283_c8 := 0;
    CONST num bStarCf6_t283_c8 := 4;
    CONST num bStarCfx_t283_c8 := 0;

    CONST num bStarCf1_t284_c2 := 0;
    CONST num bStarCf4_t284_c2 := 0;
    CONST num bStarCf6_t284_c2 := -4;
    CONST num bStarCfx_t284_c2 := 0;

    CONST num bStarCf1_t284_c3 := 0;
    CONST num bStarCf4_t284_c3 := 4;
    CONST num bStarCf6_t284_c3 := -4;
    CONST num bStarCfx_t284_c3 := 0;

    CONST num bStarCf1_t286_c2 := 0;
    CONST num bStarCf4_t286_c2 := 0;
    CONST num bStarCf6_t286_c2 := -4;
    CONST num bStarCfx_t286_c2 := 0;

    CONST num bStarCf1_t288_c5 := 0;
    CONST num bStarCf4_t288_c5 := 0;
    CONST num bStarCf6_t288_c5 := 0;
    CONST num bStarCfx_t288_c5 := 0;

    CONST num bStarCf1_t290_c5 := 0;
    CONST num bStarCf4_t290_c5 := 0;
    CONST num bStarCf6_t290_c5 := 0;
    CONST num bStarCfx_t290_c5 := 0;

    CONST num bStarCf1_t290_c6 := 0;
    CONST num bStarCf4_t290_c6 := 4;
    CONST num bStarCf6_t290_c6 := 0;
    CONST num bStarCfx_t290_c6 := 0;

    CONST num bStarCf1_t291_c5 := 0;
    CONST num bStarCf4_t291_c5 := 0;
    CONST num bStarCf6_t291_c5 := 0;
    CONST num bStarCfx_t291_c5 := 0;

    CONST num bStarCf1_t293_c5 := 0;
    CONST num bStarCf4_t293_c5 := 0;
    CONST num bStarCf6_t293_c5 := 0;
    CONST num bStarCfx_t293_c5 := 0;

    CONST num bStarCf1_t294_c3 := 0;
    CONST num bStarCf4_t294_c3 := 4;
    CONST num bStarCf6_t294_c3 := -4;
    CONST num bStarCfx_t294_c3 := 0;

    CONST num bStarCf1_t295_c5 := 0;
    CONST num bStarCf4_t295_c5 := 0;
    CONST num bStarCf6_t295_c5 := 0;
    CONST num bStarCfx_t295_c5 := 0;

    CONST num bStarCf1_t296_c5 := 0;
    CONST num bStarCf4_t296_c5 := 0;
    CONST num bStarCf6_t296_c5 := 0;
    CONST num bStarCfx_t296_c5 := 0;

    CONST num bStarCf1_t297_c2 := 0;
    CONST num bStarCf4_t297_c2 := 0;
    CONST num bStarCf6_t297_c2 := -4;
    CONST num bStarCfx_t297_c2 := 0;

    CONST num bStarCf1_t297_c5 := 0;
    CONST num bStarCf4_t297_c5 := 0;
    CONST num bStarCf6_t297_c5 := 0;
    CONST num bStarCfx_t297_c5 := 0;

    CONST num bStarCf1_t298_c2 := 0;
    CONST num bStarCf4_t298_c2 := 0;
    CONST num bStarCf6_t298_c2 := -4;
    CONST num bStarCfx_t298_c2 := 0;

    CONST num bStarCf1_t299_c5 := 0;
    CONST num bStarCf4_t299_c5 := 0;
    CONST num bStarCf6_t299_c5 := 0;
    CONST num bStarCfx_t299_c5 := 0;

    CONST num bStarCf1_t299_c8 := 0;
    CONST num bStarCf4_t299_c8 := 0;
    CONST num bStarCf6_t299_c8 := 4;
    CONST num bStarCfx_t299_c8 := 0;

    CONST num bStarCf1_t301_c5 := 0;
    CONST num bStarCf4_t301_c5 := 0;
    CONST num bStarCf6_t301_c5 := 0;
    CONST num bStarCfx_t301_c5 := 0;

    CONST num bStarCf1_t303_c5 := 0;
    CONST num bStarCf4_t303_c5 := 0;
    CONST num bStarCf6_t303_c5 := 0;
    CONST num bStarCfx_t303_c5 := 0;

    CONST num bStarCf1_t306_c2 := 0;
    CONST num bStarCf4_t306_c2 := 0;
    CONST num bStarCf6_t306_c2 := -4;
    CONST num bStarCfx_t306_c2 := 0;

    CONST num bStarCf1_t306_c5 := 0;
    CONST num bStarCf4_t306_c5 := 0;
    CONST num bStarCf6_t306_c5 := 0;
    CONST num bStarCfx_t306_c5 := 0;

    CONST num bStarCf1_t307_c5 := 0;
    CONST num bStarCf4_t307_c5 := 0;
    CONST num bStarCf6_t307_c5 := 0;
    CONST num bStarCfx_t307_c5 := 0;

    CONST num bStarCf1_t308_c4 := 0;
    CONST num bStarCf4_t308_c4 := -4;
    CONST num bStarCf6_t308_c4 := 0;
    CONST num bStarCfx_t308_c4 := 0;

    CONST num bStarCf1_t308_c5 := 0;
    CONST num bStarCf4_t308_c5 := 0;
    CONST num bStarCf6_t308_c5 := 0;
    CONST num bStarCfx_t308_c5 := 0;

    CONST num bStarCf1_t311_c4 := 0;
    CONST num bStarCf4_t311_c4 := -4;
    CONST num bStarCf6_t311_c4 := 0;
    CONST num bStarCfx_t311_c4 := 0;

    CONST num bStarCf1_t316_c5 := 0;
    CONST num bStarCf4_t316_c5 := 0;
    CONST num bStarCf6_t316_c5 := 0;
    CONST num bStarCfx_t316_c5 := 0;

    CONST num bStarCf1_t317_c5 := 0;
    CONST num bStarCf4_t317_c5 := 0;
    CONST num bStarCf6_t317_c5 := 0;
    CONST num bStarCfx_t317_c5 := 0;

    CONST num bStarCf1_t317_c8 := 0;
    CONST num bStarCf4_t317_c8 := 0;
    CONST num bStarCf6_t317_c8 := 4;
    CONST num bStarCfx_t317_c8 := 0;

    CONST num bStarCf1_t319_c2 := 0;
    CONST num bStarCf4_t319_c2 := 0;
    CONST num bStarCf6_t319_c2 := -4;
    CONST num bStarCfx_t319_c2 := 0;

    CONST num bStarCf1_t320_c5 := 0;
    CONST num bStarCf4_t320_c5 := 0;
    CONST num bStarCf6_t320_c5 := 0;
    CONST num bStarCfx_t320_c5 := 0;

    CONST num bStarCf1_t322_c6 := 0;
    CONST num bStarCf4_t322_c6 := 4;
    CONST num bStarCf6_t322_c6 := 0;
    CONST num bStarCfx_t322_c6 := 0;

    CONST num bStarCf1_t323_c1 := 0;
    CONST num bStarCf4_t323_c1 := -4;
    CONST num bStarCf6_t323_c1 := -4;
    CONST num bStarCfx_t323_c1 := 0;

    CONST num bStarCf1_t325_c2 := 0;
    CONST num bStarCf4_t325_c2 := 0;
    CONST num bStarCf6_t325_c2 := -4;
    CONST num bStarCfx_t325_c2 := 0;

    CONST num bStarCf1_t325_c5 := 0;
    CONST num bStarCf4_t325_c5 := 0;
    CONST num bStarCf6_t325_c5 := 0;
    CONST num bStarCfx_t325_c5 := 0;

    CONST num bStarCf1_t326_c5 := 0;
    CONST num bStarCf4_t326_c5 := 0;
    CONST num bStarCf6_t326_c5 := 0;
    CONST num bStarCfx_t326_c5 := 0;

    CONST num bStarCf1_t326_c8 := 0;
    CONST num bStarCf4_t326_c8 := 0;
    CONST num bStarCf6_t326_c8 := 4;
    CONST num bStarCfx_t326_c8 := 0;

    CONST num bStarCf1_t327_c5 := 0;
    CONST num bStarCf4_t327_c5 := 0;
    CONST num bStarCf6_t327_c5 := 0;
    CONST num bStarCfx_t327_c5 := 0;

    CONST num bStarCf1_t328_c2 := 0;
    CONST num bStarCf4_t328_c2 := 0;
    CONST num bStarCf6_t328_c2 := -4;
    CONST num bStarCfx_t328_c2 := 0;

    CONST num bStarCf1_t330_c2 := 0;
    CONST num bStarCf4_t330_c2 := 0;
    CONST num bStarCf6_t330_c2 := -4;
    CONST num bStarCfx_t330_c2 := 0;

    CONST num bStarCf1_t330_c5 := 0;
    CONST num bStarCf4_t330_c5 := 0;
    CONST num bStarCf6_t330_c5 := 0;
    CONST num bStarCfx_t330_c5 := 0;

    CONST num bStarCf1_t331_c2 := 0;
    CONST num bStarCf4_t331_c2 := 0;
    CONST num bStarCf6_t331_c2 := -4;
    CONST num bStarCfx_t331_c2 := 0;

    CONST num bStarCf1_t331_c5 := 0;
    CONST num bStarCf4_t331_c5 := 0;
    CONST num bStarCf6_t331_c5 := 0;
    CONST num bStarCfx_t331_c5 := 0;

    CONST num bStarCf1_t336_c5 := 0;
    CONST num bStarCf4_t336_c5 := 0;
    CONST num bStarCf6_t336_c5 := 0;
    CONST num bStarCfx_t336_c5 := 0;

    CONST num bStarCf1_t336_c8 := 0;
    CONST num bStarCf4_t336_c8 := 0;
    CONST num bStarCf6_t336_c8 := 4;
    CONST num bStarCfx_t336_c8 := 0;

    CONST num bStarCf1_t337_c2 := 0;
    CONST num bStarCf4_t337_c2 := 0;
    CONST num bStarCf6_t337_c2 := -4;
    CONST num bStarCfx_t337_c2 := 0;

    CONST num bStarCf1_t337_c5 := 0;
    CONST num bStarCf4_t337_c5 := 0;
    CONST num bStarCf6_t337_c5 := 0;
    CONST num bStarCfx_t337_c5 := 0;

    CONST num bStarCf1_t338_c4 := 0;
    CONST num bStarCf4_t338_c4 := -4;
    CONST num bStarCf6_t338_c4 := 0;
    CONST num bStarCfx_t338_c4 := 0;

    CONST num bStarCf1_t338_c7 := 0;
    CONST num bStarCf4_t338_c7 := -4;
    CONST num bStarCf6_t338_c7 := 4;
    CONST num bStarCfx_t338_c7 := 0;

    CONST num bStarCf1_t339_c8 := 0;
    CONST num bStarCf4_t339_c8 := 0;
    CONST num bStarCf6_t339_c8 := 4;
    CONST num bStarCfx_t339_c8 := 0;

    CONST num bStarCf1_t340_c5 := 0;
    CONST num bStarCf4_t340_c5 := 0;
    CONST num bStarCf6_t340_c5 := 0;
    CONST num bStarCfx_t340_c5 := 0;

    CONST num bStarCf1_t340_c6 := 0;
    CONST num bStarCf4_t340_c6 := 4;
    CONST num bStarCf6_t340_c6 := 0;
    CONST num bStarCfx_t340_c6 := 0;

    CONST num bStarCf1_t341_c5 := 0;
    CONST num bStarCf4_t341_c5 := 0;
    CONST num bStarCf6_t341_c5 := 0;
    CONST num bStarCfx_t341_c5 := 0;

    CONST num bStarCf1_t342_c5 := 0;
    CONST num bStarCf4_t342_c5 := 0;
    CONST num bStarCf6_t342_c5 := 0;
    CONST num bStarCfx_t342_c5 := 0;

    CONST num bStarCf1_t344_c2 := 0;
    CONST num bStarCf4_t344_c2 := 0;
    CONST num bStarCf6_t344_c2 := -4;
    CONST num bStarCfx_t344_c2 := 0;

    CONST num bStarCf1_t344_c5 := 0;
    CONST num bStarCf4_t344_c5 := 0;
    CONST num bStarCf6_t344_c5 := 0;
    CONST num bStarCfx_t344_c5 := 0;

    CONST num bStarCf1_t345_c7 := 0;
    CONST num bStarCf4_t345_c7 := -4;
    CONST num bStarCf6_t345_c7 := 4;
    CONST num bStarCfx_t345_c7 := 0;

    CONST num bStarCf1_t346_c2 := 0;
    CONST num bStarCf4_t346_c2 := 0;
    CONST num bStarCf6_t346_c2 := -4;
    CONST num bStarCfx_t346_c2 := 0;

    CONST num bStarCf1_t346_c5 := 0;
    CONST num bStarCf4_t346_c5 := 0;
    CONST num bStarCf6_t346_c5 := 0;
    CONST num bStarCfx_t346_c5 := 0;

    CONST num bStarCf1_t347_c4 := 0;
    CONST num bStarCf4_t347_c4 := -4;
    CONST num bStarCf6_t347_c4 := 0;
    CONST num bStarCfx_t347_c4 := 0;

    CONST num bStarCf1_t350_c4 := 0;
    CONST num bStarCf4_t350_c4 := -4;
    CONST num bStarCf6_t350_c4 := 0;
    CONST num bStarCfx_t350_c4 := 0;

    CONST num bStarCf1_t353_c2 := 0;
    CONST num bStarCf4_t353_c2 := 0;
    CONST num bStarCf6_t353_c2 := -4;
    CONST num bStarCfx_t353_c2 := 0;

    CONST num bStarCf1_t353_c5 := 0;
    CONST num bStarCf4_t353_c5 := 0;
    CONST num bStarCf6_t353_c5 := 0;
    CONST num bStarCfx_t353_c5 := 0;

    CONST num bStarCf1_t354_c5 := 0;
    CONST num bStarCf4_t354_c5 := 0;
    CONST num bStarCf6_t354_c5 := 0;
    CONST num bStarCfx_t354_c5 := 0;

    CONST num bStarCf1_t357_c4 := 0;
    CONST num bStarCf4_t357_c4 := -4;
    CONST num bStarCf6_t357_c4 := 0;
    CONST num bStarCfx_t357_c4 := 0;

    CONST num bStarCf1_t357_c7 := 0;
    CONST num bStarCf4_t357_c7 := -4;
    CONST num bStarCf6_t357_c7 := 4;
    CONST num bStarCfx_t357_c7 := 0;

    CONST num bStarCf1_t360_c5 := 0;
    CONST num bStarCf4_t360_c5 := 0;
    CONST num bStarCf6_t360_c5 := 0;
    CONST num bStarCfx_t360_c5 := 0;

    CONST num bStarCf1_t361_c5 := 0;
    CONST num bStarCf4_t361_c5 := 0;
    CONST num bStarCf6_t361_c5 := 0;
    CONST num bStarCfx_t361_c5 := 0;

    CONST num bStarCf1_t362_c4 := 0;
    CONST num bStarCf4_t362_c4 := -4;
    CONST num bStarCf6_t362_c4 := 0;
    CONST num bStarCfx_t362_c4 := 0;

    CONST num bStarCf1_t363_c5 := 0;
    CONST num bStarCf4_t363_c5 := 0;
    CONST num bStarCf6_t363_c5 := 0;
    CONST num bStarCfx_t363_c5 := 0;

    CONST num bStarCf1_t364_c4 := 0;
    CONST num bStarCf4_t364_c4 := -4;
    CONST num bStarCf6_t364_c4 := 0;
    CONST num bStarCfx_t364_c4 := 0;

    CONST num bStarCf1_t368_c4 := 0;
    CONST num bStarCf4_t368_c4 := -4;
    CONST num bStarCf6_t368_c4 := 0;
    CONST num bStarCfx_t368_c4 := 0;

    CONST num bStarCf1_t374_c5 := 0;
    CONST num bStarCf4_t374_c5 := 0;
    CONST num bStarCf6_t374_c5 := 0;
    CONST num bStarCfx_t374_c5 := 0;

    CONST num bStarCf1_t383_c2 := 0;
    CONST num bStarCf4_t383_c2 := 0;
    CONST num bStarCf6_t383_c2 := -4;
    CONST num bStarCfx_t383_c2 := 0;

    CONST num bStarCf1_t389_c5 := 0;
    CONST num bStarCf4_t389_c5 := 0;
    CONST num bStarCf6_t389_c5 := 0;
    CONST num bStarCfx_t389_c5 := 0;

    CONST num bStarCf1_t392_c2 := 0;
    CONST num bStarCf4_t392_c2 := 0;
    CONST num bStarCf6_t392_c2 := -4;
    CONST num bStarCfx_t392_c2 := 0;

    CONST num bStarCf1_t392_c5 := 0;
    CONST num bStarCf4_t392_c5 := 0;
    CONST num bStarCf6_t392_c5 := 0;
    CONST num bStarCfx_t392_c5 := 0;

    CONST num bStarCf1_t393_c5 := 0;
    CONST num bStarCf4_t393_c5 := 0;
    CONST num bStarCf6_t393_c5 := 0;
    CONST num bStarCfx_t393_c5 := 0;

    CONST num bStarCf1_t393_c8 := 0;
    CONST num bStarCf4_t393_c8 := 0;
    CONST num bStarCf6_t393_c8 := 4;
    CONST num bStarCfx_t393_c8 := 0;

    CONST num bStarCf1_t394_c7 := 0;
    CONST num bStarCf4_t394_c7 := -4;
    CONST num bStarCf6_t394_c7 := 4;
    CONST num bStarCfx_t394_c7 := 0;

    CONST num bStarCf1_t396_c7 := 0;
    CONST num bStarCf4_t396_c7 := -4;
    CONST num bStarCf6_t396_c7 := 4;
    CONST num bStarCfx_t396_c7 := 0;

    CONST num bStarCf1_t397_c5 := 0;
    CONST num bStarCf4_t397_c5 := 0;
    CONST num bStarCf6_t397_c5 := 0;
    CONST num bStarCfx_t397_c5 := 0;

    CONST num bStarCf1_t398_c4 := 0;
    CONST num bStarCf4_t398_c4 := -4;
    CONST num bStarCf6_t398_c4 := 0;
    CONST num bStarCfx_t398_c4 := 0;

    CONST num bStarCf1_t399_c8 := 0;
    CONST num bStarCf4_t399_c8 := 0;
    CONST num bStarCf6_t399_c8 := 4;
    CONST num bStarCfx_t399_c8 := 0;

    CONST num bStarCf1_t402_c5 := 0;
    CONST num bStarCf4_t402_c5 := 0;
    CONST num bStarCf6_t402_c5 := 0;
    CONST num bStarCfx_t402_c5 := 0;

    CONST num bStarCf1_t404_c2 := 0;
    CONST num bStarCf4_t404_c2 := 0;
    CONST num bStarCf6_t404_c2 := -4;
    CONST num bStarCfx_t404_c2 := 0;

    CONST num bStarCf1_t404_c5 := 0;
    CONST num bStarCf4_t404_c5 := 0;
    CONST num bStarCf6_t404_c5 := 0;
    CONST num bStarCfx_t404_c5 := 0;

    CONST num bStarCf1_t405_c5 := 0;
    CONST num bStarCf4_t405_c5 := 0;
    CONST num bStarCf6_t405_c5 := 0;
    CONST num bStarCfx_t405_c5 := 0;

    CONST num bStarCf1_t406_c5 := 0;
    CONST num bStarCf4_t406_c5 := 0;
    CONST num bStarCf6_t406_c5 := 0;
    CONST num bStarCfx_t406_c5 := 0;

    CONST num bStarCf1_t406_c8 := 0;
    CONST num bStarCf4_t406_c8 := 0;
    CONST num bStarCf6_t406_c8 := 4;
    CONST num bStarCfx_t406_c8 := 0;

    CONST num bStarCf1_t408_c5 := 0;
    CONST num bStarCf4_t408_c5 := 0;
    CONST num bStarCf6_t408_c5 := 0;
    CONST num bStarCfx_t408_c5 := 0;

    CONST num bStarCf1_t409_c5 := 0;
    CONST num bStarCf4_t409_c5 := 0;
    CONST num bStarCf6_t409_c5 := 0;
    CONST num bStarCfx_t409_c5 := 0;

    CONST num bStarCf1_t409_c8 := 0;
    CONST num bStarCf4_t409_c8 := 0;
    CONST num bStarCf6_t409_c8 := 4;
    CONST num bStarCfx_t409_c8 := 0;

    CONST num bStarCf1_t411_c1 := 0;
    CONST num bStarCf4_t411_c1 := -4;
    CONST num bStarCf6_t411_c1 := -4;
    CONST num bStarCfx_t411_c1 := 0;

    CONST num bStarCf1_t413_c6 := 0;
    CONST num bStarCf4_t413_c6 := 4;
    CONST num bStarCf6_t413_c6 := 0;
    CONST num bStarCfx_t413_c6 := 0;

    CONST num bStarCf1_t414_c2 := 0;
    CONST num bStarCf4_t414_c2 := 0;
    CONST num bStarCf6_t414_c2 := -4;
    CONST num bStarCfx_t414_c2 := 0;

    CONST num bStarCf1_t418_c4 := 0;
    CONST num bStarCf4_t418_c4 := -4;
    CONST num bStarCf6_t418_c4 := 0;
    CONST num bStarCfx_t418_c4 := 0;

    CONST num bStarCf1_t418_c5 := 0;
    CONST num bStarCf4_t418_c5 := 0;
    CONST num bStarCf6_t418_c5 := 0;
    CONST num bStarCfx_t418_c5 := 0;

    CONST num bStarCf1_t419_c2 := 0;
    CONST num bStarCf4_t419_c2 := 0;
    CONST num bStarCf6_t419_c2 := -4;
    CONST num bStarCfx_t419_c2 := 0;

    CONST num bStarCf1_t424_c5 := 0;
    CONST num bStarCf4_t424_c5 := 0;
    CONST num bStarCf6_t424_c5 := 0;
    CONST num bStarCfx_t424_c5 := 0;

    CONST num bStarCf1_t425_c5 := 0;
    CONST num bStarCf4_t425_c5 := 0;
    CONST num bStarCf6_t425_c5 := 0;
    CONST num bStarCfx_t425_c5 := 0;

    CONST num bStarCf1_t426_c1 := 0;
    CONST num bStarCf4_t426_c1 := -4;
    CONST num bStarCf6_t426_c1 := -4;
    CONST num bStarCfx_t426_c1 := 0;

    CONST num bStarCf1_t428_c5 := 0;
    CONST num bStarCf4_t428_c5 := 0;
    CONST num bStarCf6_t428_c5 := 0;
    CONST num bStarCfx_t428_c5 := 0;

    CONST num bStarCf1_t429_c8 := 0;
    CONST num bStarCf4_t429_c8 := 0;
    CONST num bStarCf6_t429_c8 := 4;
    CONST num bStarCfx_t429_c8 := 0;

    CONST num bStarCf1_t438_c5 := 0;
    CONST num bStarCf4_t438_c5 := 0;
    CONST num bStarCf6_t438_c5 := 0;
    CONST num bStarCfx_t438_c5 := 0;

    CONST num bStarCf1_t440_c1 := 0;
    CONST num bStarCf4_t440_c1 := -4;
    CONST num bStarCf6_t440_c1 := -4;
    CONST num bStarCfx_t440_c1 := 0;

    CONST num bStarCf1_t440_c4 := 0;
    CONST num bStarCf4_t440_c4 := -4;
    CONST num bStarCf6_t440_c4 := 0;
    CONST num bStarCfx_t440_c4 := 0;

    CONST num bStarCf1_t442_c5 := 0;
    CONST num bStarCf4_t442_c5 := 0;
    CONST num bStarCf6_t442_c5 := 0;
    CONST num bStarCfx_t442_c5 := 0;

    CONST num bStarCf1_t443_c4 := 0;
    CONST num bStarCf4_t443_c4 := -4;
    CONST num bStarCf6_t443_c4 := 0;
    CONST num bStarCfx_t443_c4 := 0;

    CONST num bStarCf1_t444_c4 := 0;
    CONST num bStarCf4_t444_c4 := -4;
    CONST num bStarCf6_t444_c4 := 0;
    CONST num bStarCfx_t444_c4 := 0;

    CONST num bStarCf1_t444_c7 := 0;
    CONST num bStarCf4_t444_c7 := -4;
    CONST num bStarCf6_t444_c7 := 4;
    CONST num bStarCfx_t444_c7 := 0;

    CONST num bStarCf1_t446_c1 := 0;
    CONST num bStarCf4_t446_c1 := -4;
    CONST num bStarCf6_t446_c1 := -4;
    CONST num bStarCfx_t446_c1 := 0;

    CONST num bStarCf1_t446_c2 := 0;
    CONST num bStarCf4_t446_c2 := 0;
    CONST num bStarCf6_t446_c2 := -4;
    CONST num bStarCfx_t446_c2 := 0;

    CONST num bStarCf1_t448_c5 := 0;
    CONST num bStarCf4_t448_c5 := 0;
    CONST num bStarCf6_t448_c5 := 0;
    CONST num bStarCfx_t448_c5 := 0;

    CONST num bStarCf1_t449_c1 := 0;
    CONST num bStarCf4_t449_c1 := -4;
    CONST num bStarCf6_t449_c1 := -4;
    CONST num bStarCfx_t449_c1 := 0;

    CONST num bStarCf1_t449_c2 := 0;
    CONST num bStarCf4_t449_c2 := 0;
    CONST num bStarCf6_t449_c2 := -4;
    CONST num bStarCfx_t449_c2 := 0;

    CONST num bStarCf1_t450_c4 := 0;
    CONST num bStarCf4_t450_c4 := -4;
    CONST num bStarCf6_t450_c4 := 0;
    CONST num bStarCfx_t450_c4 := 0;

    CONST num bStarCf1_t450_c5 := 0;
    CONST num bStarCf4_t450_c5 := 0;
    CONST num bStarCf6_t450_c5 := 0;
    CONST num bStarCfx_t450_c5 := 0;

    CONST num bStarCf1_t451_c4 := 0;
    CONST num bStarCf4_t451_c4 := -4;
    CONST num bStarCf6_t451_c4 := 0;
    CONST num bStarCfx_t451_c4 := 0;

    CONST num bStarCf1_t452_c2 := 0;
    CONST num bStarCf4_t452_c2 := 0;
    CONST num bStarCf6_t452_c2 := -4;
    CONST num bStarCfx_t452_c2 := 0;

    CONST num bStarCf1_t455_c4 := 0;
    CONST num bStarCf4_t455_c4 := -4;
    CONST num bStarCf6_t455_c4 := 0;
    CONST num bStarCfx_t455_c4 := 0;

    CONST num bStarCf1_t455_c5 := 0;
    CONST num bStarCf4_t455_c5 := 0;
    CONST num bStarCf6_t455_c5 := 0;
    CONST num bStarCfx_t455_c5 := 0;

    CONST num bStarCf1_t461_c4 := 0;
    CONST num bStarCf4_t461_c4 := -4;
    CONST num bStarCf6_t461_c4 := 0;
    CONST num bStarCfx_t461_c4 := 0;

    CONST num bStarCf1_t461_c5 := 0;
    CONST num bStarCf4_t461_c5 := 0;
    CONST num bStarCf6_t461_c5 := 0;
    CONST num bStarCfx_t461_c5 := 0;

    CONST num bStarCf1_t462_c2 := 0;
    CONST num bStarCf4_t462_c2 := 0;
    CONST num bStarCf6_t462_c2 := -4;
    CONST num bStarCfx_t462_c2 := 0;

    CONST num bStarCf1_t463_c2 := 0;
    CONST num bStarCf4_t463_c2 := 0;
    CONST num bStarCf6_t463_c2 := -4;
    CONST num bStarCfx_t463_c2 := 0;

    CONST num bStarCf1_t465_c5 := 0;
    CONST num bStarCf4_t465_c5 := 0;
    CONST num bStarCf6_t465_c5 := 0;
    CONST num bStarCfx_t465_c5 := 0;

    CONST num bStarCf1_t467_c8 := 0;
    CONST num bStarCf4_t467_c8 := 0;
    CONST num bStarCf6_t467_c8 := 4;
    CONST num bStarCfx_t467_c8 := 0;

    CONST num bStarCf1_t468_c4 := 0;
    CONST num bStarCf4_t468_c4 := -4;
    CONST num bStarCf6_t468_c4 := 0;
    CONST num bStarCfx_t468_c4 := 0;

    CONST num bStarCf1_t468_c7 := 0;
    CONST num bStarCf4_t468_c7 := -4;
    CONST num bStarCf6_t468_c7 := 4;
    CONST num bStarCfx_t468_c7 := 0;

    CONST num bStarCf1_t469_c9 := 0;
    CONST num bStarCf4_t469_c9 := 4;
    CONST num bStarCf6_t469_c9 := 4;
    CONST num bStarCfx_t469_c9 := 0;

    CONST num bStarCf1_t470_c1 := 0;
    CONST num bStarCf4_t470_c1 := -4;
    CONST num bStarCf6_t470_c1 := -4;
    CONST num bStarCfx_t470_c1 := 0;

    CONST num bStarCf1_t470_c4 := 0;
    CONST num bStarCf4_t470_c4 := -4;
    CONST num bStarCf6_t470_c4 := 0;
    CONST num bStarCfx_t470_c4 := 0;

    CONST num bStarCf1_t472_c4 := 0;
    CONST num bStarCf4_t472_c4 := -4;
    CONST num bStarCf6_t472_c4 := 0;
    CONST num bStarCfx_t472_c4 := 0;

    CONST num bStarCf1_t472_c5 := 0;
    CONST num bStarCf4_t472_c5 := 0;
    CONST num bStarCf6_t472_c5 := 0;
    CONST num bStarCfx_t472_c5 := 0;

    CONST num bStarCf1_t473_c4 := 0;
    CONST num bStarCf4_t473_c4 := -4;
    CONST num bStarCf6_t473_c4 := 0;
    CONST num bStarCfx_t473_c4 := 0;

    CONST num bStarCf1_t474_c4 := 0;
    CONST num bStarCf4_t474_c4 := -4;
    CONST num bStarCf6_t474_c4 := 0;
    CONST num bStarCfx_t474_c4 := 0;

    CONST num bStarCf1_t474_c5 := 0;
    CONST num bStarCf4_t474_c5 := 0;
    CONST num bStarCf6_t474_c5 := 0;
    CONST num bStarCfx_t474_c5 := 0;

    CONST num bStarCf1_t475_c2 := 0;
    CONST num bStarCf4_t475_c2 := 0;
    CONST num bStarCf6_t475_c2 := -4;
    CONST num bStarCfx_t475_c2 := 0;

    CONST num bStarCf1_t477_c4 := 0;
    CONST num bStarCf4_t477_c4 := -4;
    CONST num bStarCf6_t477_c4 := 0;
    CONST num bStarCfx_t477_c4 := 0;

    CONST num bStarCf1_t479_c7 := 0;
    CONST num bStarCf4_t479_c7 := -4;
    CONST num bStarCf6_t479_c7 := 4;
    CONST num bStarCfx_t479_c7 := 0;

    CONST num bStarCf1_t481_c2 := 0;
    CONST num bStarCf4_t481_c2 := 0;
    CONST num bStarCf6_t481_c2 := -4;
    CONST num bStarCfx_t481_c2 := 0;

    CONST num bStarCf1_t482_c2 := 0;
    CONST num bStarCf4_t482_c2 := 0;
    CONST num bStarCf6_t482_c2 := -4;
    CONST num bStarCfx_t482_c2 := 0;

    CONST num bStarCf1_t483_c4 := 0;
    CONST num bStarCf4_t483_c4 := -4;
    CONST num bStarCf6_t483_c4 := 0;
    CONST num bStarCfx_t483_c4 := 0;

    CONST num bStarCf1_t484_c4 := 0;
    CONST num bStarCf4_t484_c4 := -4;
    CONST num bStarCf6_t484_c4 := 0;
    CONST num bStarCfx_t484_c4 := 0;

    CONST num bStarCf1_t484_c7 := 0;
    CONST num bStarCf4_t484_c7 := -4;
    CONST num bStarCf6_t484_c7 := 4;
    CONST num bStarCfx_t484_c7 := 0;

    CONST num bStarCf1_t485_c2 := 0;
    CONST num bStarCf4_t485_c2 := 0;
    CONST num bStarCf6_t485_c2 := -4;
    CONST num bStarCfx_t485_c2 := 0;

    CONST num bStarCf1_t485_c5 := 0;
    CONST num bStarCf4_t485_c5 := 0;
    CONST num bStarCf6_t485_c5 := 0;
    CONST num bStarCfx_t485_c5 := 0;

    CONST num bStarCf1_t486_c5 := 0;
    CONST num bStarCf4_t486_c5 := 0;
    CONST num bStarCf6_t486_c5 := 0;
    CONST num bStarCfx_t486_c5 := 0;

    CONST num bStarCf1_t488_c5 := 0;
    CONST num bStarCf4_t488_c5 := 0;
    CONST num bStarCf6_t488_c5 := 0;
    CONST num bStarCfx_t488_c5 := 0;

    CONST num bStarCf1_t489_c4 := 0;
    CONST num bStarCf4_t489_c4 := -4;
    CONST num bStarCf6_t489_c4 := 0;
    CONST num bStarCfx_t489_c4 := 0;

    CONST num bStarCf1_t489_c5 := 0;
    CONST num bStarCf4_t489_c5 := 0;
    CONST num bStarCf6_t489_c5 := 0;
    CONST num bStarCfx_t489_c5 := 0;

    CONST num bStarCf1_t490_c4 := 0;
    CONST num bStarCf4_t490_c4 := -4;
    CONST num bStarCf6_t490_c4 := 0;
    CONST num bStarCfx_t490_c4 := 0;

    CONST num bStarCf1_t491_c5 := 0;
    CONST num bStarCf4_t491_c5 := 0;
    CONST num bStarCf6_t491_c5 := 0;
    CONST num bStarCfx_t491_c5 := 0;

    CONST num bStarCf1_t493_c3 := 0;
    CONST num bStarCf4_t493_c3 := 4;
    CONST num bStarCf6_t493_c3 := -4;
    CONST num bStarCfx_t493_c3 := 0;

    CONST num bStarCf1_t493_c8 := 0;
    CONST num bStarCf4_t493_c8 := 0;
    CONST num bStarCf6_t493_c8 := 4;
    CONST num bStarCfx_t493_c8 := 0;

    CONST num bStarCf1_t495_c1 := 0;
    CONST num bStarCf4_t495_c1 := -4;
    CONST num bStarCf6_t495_c1 := -4;
    CONST num bStarCfx_t495_c1 := 0;

    CONST num bStarCf1_t495_c4 := 0;
    CONST num bStarCf4_t495_c4 := -4;
    CONST num bStarCf6_t495_c4 := 0;
    CONST num bStarCfx_t495_c4 := 0;

    CONST num bStarCf1_t496_c5 := 0;
    CONST num bStarCf4_t496_c5 := 0;
    CONST num bStarCf6_t496_c5 := 0;
    CONST num bStarCfx_t496_c5 := 0;

    CONST num bStarCf1_t498_c2 := 0;
    CONST num bStarCf4_t498_c2 := 0;
    CONST num bStarCf6_t498_c2 := -4;
    CONST num bStarCfx_t498_c2 := 0;

ENDMODULE
